INTERFACE ITF_Group2_HMI_Connector_View EXTENDS ITF_BaseGroupElement_HMI_Connector_View

END_INTERFACE

(* stored: Version 1.1.0.1
   Itf ITF_Group2_HMI_Connector_View: Id {9082d202-9c92-0399-1b85-ebbfbf8dcd9a} *)
